FUNCTION_BLOCK Robot_Weld

VAR_INPUT
	Robot_1_In			:	Weld_Robot;
	Part_Unload_Comp	:	BOOL;
END_VAR

VAR_OUTPUT
	Robot_1_Out			:	Weld_Robot;	
END_VAR

VAR
	Weld_Delay			:	TON;
END_VAR

CASE Robot_1_In.i_Prg_No OF
	101:
		IF (Robot_1_In.i_Area_Ok AND Robot_1_In.i_Start) THEN
		Robot_1_In.i_Home := FALSE;
		Weld_Delay(IN:= Robot_1_In.i_Start, PT:= T#1S, Q=> , ET=> );
		IF Weld_Delay.Q THEN
		Robot_1_Out.o_Weld_Comp := TRUE;
		Robot_1_In.i_Home := TRUE;
		END_IF
		END_IF
		IF (Robot_1_In.i_Home AND Part_Unload_Comp) THEN
		Robot_1_Out.o_Weld_Comp := FALSE;	
		END_IF
		Robot_1_In.i_Prg_No := 101;
	102:
		IF (Robot_1_In.i_Area_Ok AND Robot_1_In.i_Start) THEN
		Robot_1_In.i_Home := FALSE;
		Weld_Delay(IN:= Robot_1_In.i_Start, PT:= T#1S, Q=> , ET=> );
		IF Weld_Delay.Q THEN
		Robot_1_Out.o_Weld_Comp := TRUE;
		Robot_1_In.i_Home := TRUE;
		END_IF
		END_IF
		IF (Robot_1_In.i_Home AND Part_Unload_Comp) THEN
		Robot_1_Out.o_Weld_Comp := FALSE;	
		END_IF
		Robot_1_In.i_Prg_No := 102;
END_CASE

END_FUNCTION_BLOCK

(* stored: Version 1.1.0.1, ProductVersion 3.1.4024.16
   POU Robot_Weld: Id {a7105986-11fb-407c-b397-ca5ac0e537ce}, SpecialFunc None *)
